{attribute 'linkalways'} 
{attribute 'no_explicit_call' := 'This FB is a CLASS and must be accessed using methods or properties'}
{attribute 'enable_dynamic_creation'}
FUNCTION_BLOCK Node_F_VN_CalibrateCameraPlanar EXTENDS VisionNode
VAR
    ipSrcImage : _ITcVnImage;
    aMarkerPositions : _TcVnArray4_Point2_REAL;
    aTransformationMatrix : _TcVnMatrix3x3_LREAL;
    hrPrev : _HRESULT(S_OK);
	hresult : _HRESULT(S_OK);
END_VAR

METHOD PUBLIC  Clone : I_Node
VAR
	pNode : POINTER TO Node_F_VN_CalibrateCameraPlanar;
END_VAR
pNode := __NEW(Node_F_VN_CalibrateCameraPlanar);
Clone := pNode^;
END_METHOD

METHOD FB_init : BOOL
VAR_INPUT
	bInitRetains : BOOL; // if TRUE, the retain variables are initialized (warm start / cold start)
	bInCopyCode : BOOL;  // if TRUE, the instance afterwards gets moved into the copy code (online change)
END_VAR
AddInput('ipSrcImage', ipSrcImage);
AddInput('aMarkerPositions', aMarkerPositions);
AddInput('hrPrev', hrPrev);
AddOutput('aTransformationMatrix', aTransformationMatrix);
AddOutput('hresult', hresult);
END_METHOD

METHOD PROTECTED OnExecute
hresult.Value := F_VN_CalibrateCameraPlanar(
    ipSrcImage := ipSrcImage.Value,
    aMarkerPositions := aMarkerPositions.Value,
    aTransformationMatrix := aTransformationMatrix.Value,
	hrPrev := hrPrev.Value);
END_METHOD

METHOD PUBLIC PreExecutionCheck
VAR_INPUT
	Check : I_PreExecutionChecks;
END_VAR
Check.IsTrue(ipSrcImage.IsValid, 'ipSrcImage must contain an image');
END_METHOD

END_FUNCTION_BLOCK

(* stored: Version 1.1.0.1, ProductVersion 3.1.4024.15
   POU Node_F_VN_CalibrateCameraPlanar: Id {91a3dcae-304b-4f80-b3a9-d5ed0366f434}, SpecialFunc None
   Folder Constructor: Id {9599f7ba-c50b-4d05-ac17-4c553abb0957}
   Method Clone: Id {f26a772e-ceaa-4c7a-bcd8-7f988b1422e5}
   Method FB_init: Id {bbabf8a2-bb0e-4ebb-b1af-db33173f171e}
   Method OnExecute: Id {0ebde6bb-31b5-4781-8157-13f9b116879d}
   Method PreExecutionCheck: Id {4a653df4-c6cd-4599-9e81-4e45984131ad} *)
